// TIA Portal V16 export
// export: Created 2022-11-14T17:35:47.4589273Z, ExportSetting WithDefaults, DisplayName Totally Integrated Automation Portal, DisplayVersion V16, DisplayName TIA Portal Version Control Interface, DisplayVersion V16, DisplayName TIA Portal Openness, DisplayVersion V16, DisplayName STEP 7 Professional, DisplayVersion V16, DisplayName STEP 7 Safety, DisplayVersion V16, DisplayName WinCC Advanced, DisplayVersion V16
DATA_BLOCK "DB239_Program11"   // DB239
{ S7_Optimized_Access := 'FALSE' }
AUTHOR : Robopac
VERSION : 0.0
// stored: AutoNumber false, IsOnlyStoredInLoadMemory false, IsWriteProtectedInAS false
   VAR RETAIN
      Program11 { S7_SetPoint := 'True'} : "DatiProgramma";
   END_VAR
BEGIN
   Program11.Wrapping := TRUE;
   Program11.TopLenght := 500;
   Program11.TopRelease := 0;
   Program11.TopDown := 0;
   Program11.Top := 4;
   Program11.PressurePTime := 0;
   Program11.LifterTime := 0;
   Program11.RevOverContrast := 1;
   Program11.RopeEndCycle := 16#02;
   Program11.Spare4 := 16#01;
   Program11.RopeTime := 1500;
   Program11.RevOverClamp := 1;
   Program11.FilmForceFinalRev := 10;
   Program11.FilmPrestretchFinalRev := 100;
   Program11.ArmSpeed := 100;
   Program11.CarriageDown4Top := 500;
   Program11.TopDownTime := 1500;
   Program11.LapsUnderTop := 0;
   Program11.Spare6 := 0;
   Program11.Spare7 := 0;
   Program11.Spare8 := 0;
   Program11.Spare9 := 0;
   Program11.Spare10 := 0;
   Program11.Spare11 := 0;
   Program11.Spare12 := 0;
   Program11.Overlap0_1 := 0;
   Program11.Height1 := 130;
   Program11.Landmark1 := FALSE;
   Program11.Lifter1 := FALSE;
   Program11.SpareBit1H1 := FALSE;
   Program11.Airblower1 := TRUE;
   Program11.NextStep1 := TRUE;
   Program11.PressureP1 := TRUE;
   Program11.SpareByte2H1 := 16#00;
   Program11.Revolution1 := 1;
   Program11.RopeUnit1_1 := 16#01;
   Program11.RopeUnit1_2 := 16#01;
   Program11.FilmForce1 := 5;
   Program11.FilmPrestretch1 := 200;
   Program11.Spare3H1 := 0;
   Program11.Spare49 := 0;
   Program11.Spare50 := 0;
   Program11.Spare51 := 0;
   Program11.Spare52 := 0;
   Program11.Spare53 := 0;
   Program11.Overlap1_2 := 0;
   Program11.Height2 := 50;
   Program11.Landmark2 := FALSE;
   Program11.Lifter2 := FALSE;
   Program11.SpareBit1H2 := FALSE;
   Program11.Airblower2 := TRUE;
   Program11.NextStep2 := TRUE;
   Program11.PressureP2 := TRUE;
   Program11.SpareByte2H2 := 16#00;
   Program11.Revolution2 := 1;
   Program11.RopeUnit2_1 := 16#01;
   Program11.RopeUnit2_2 := 16#01;
   Program11.FilmForce2 := 20;
   Program11.FilmPrestretch2 := 200;
   Program11.Spare3H2 := 0;
   Program11.Spare54 := 0;
   Program11.Spare55 := 0;
   Program11.Spare56 := 0;
   Program11.Spare57 := 0;
   Program11.Spare58 := 0;
   Program11.Overlap2_3 := 100;
   Program11.Height3 := -50;
   Program11.Landmark3 := TRUE;
   Program11.Lifter3 := FALSE;
   Program11.SpareBit1H3 := FALSE;
   Program11.Airblower3 := TRUE;
   Program11.NextStep3 := TRUE;
   Program11.PressureP3 := TRUE;
   Program11.SpareByte2H3 := 16#00;
   Program11.Revolution3 := 2;
   Program11.RopeUnit3_1 := 16#01;
   Program11.RopeUnit3_2 := 16#01;
   Program11.FilmForce3 := 30;
   Program11.FilmPrestretch3 := 200;
   Program11.Spare3H3 := 0;
   Program11.Spare59 := 0;
   Program11.Spare60 := 0;
   Program11.Spare61 := 380;
   Program11.Spare62 := 2800;
   Program11.Spare63 := 0;
   Program11.Overlap3_4 := 100;
   Program11.Height4 := 100;
   Program11.Landmark4 := FALSE;
   Program11.Lifter4 := FALSE;
   Program11.SpareBit1H4 := FALSE;
   Program11.Airblower4 := TRUE;
   Program11.NextStep4 := TRUE;
   Program11.PressureP4 := TRUE;
   Program11.SpareByte2H4 := 16#00;
   Program11.Revolution4 := 3;
   Program11.RopeUnit4_1 := 16#02;
   Program11.RopeUnit4_2 := 16#02;
   Program11.FilmForce4 := 30;
   Program11.FilmPrestretch4 := 200;
   Program11.Spare3H4 := 0;
   Program11.Spare64 := 0;
   Program11.Spare65 := 0;
   Program11.Spare66 := 0;
   Program11.Spare67 := 0;
   Program11.Spare68 := 0;
   Program11.Overlap4_5 := 0;
   Program11.Height5 := 50;
   Program11.Landmark5 := FALSE;
   Program11.Lifter5 := FALSE;
   Program11.SpareBit1H5 := FALSE;
   Program11.Airblower5 := TRUE;
   Program11.NextStep5 := FALSE;
   Program11.PressureP5 := FALSE;
   Program11.SpareByte2H5 := 16#00;
   Program11.Revolution5 := 1;
   Program11.RopeUnit5_1 := 16#01;
   Program11.RopeUnit5_2 := 16#01;
   Program11.FilmForce5 := 30;
   Program11.FilmPrestretch5 := 200;
   Program11.Spare3H5 := 0;
   Program11.Spare69 := 0;
   Program11.Spare70 := 0;
   Program11.Spare71 := 0;
   Program11.Spare72 := 0;
   Program11.Spare73 := 0;
   Program11.Overlap5_6 := 100;
   Program11.Height6 := 50;
   Program11.Landmark6 := FALSE;
   Program11.Lifter6 := FALSE;
   Program11.SpareBit1H6 := FALSE;
   Program11.Airblower6 := TRUE;
   Program11.NextStep6 := FALSE;
   Program11.PressureP6 := FALSE;
   Program11.SpareByte2H6 := 16#00;
   Program11.Revolution6 := 2;
   Program11.RopeUnit6_1 := 16#02;
   Program11.RopeUnit6_2 := 16#01;
   Program11.FilmForce6 := 20;
   Program11.FilmPrestretch6 := 200;
   Program11.Spare3H6 := 0;
   Program11.Spare74 := 0;
   Program11.Spare75 := 0;
   Program11.Spare76 := 0;
   Program11.Spare77 := 0;
   Program11.Spare78 := 0;
   Program11.Overlap6_7 := 0;
   Program11.Height7 := 0;
   Program11.Landmark7 := FALSE;
   Program11.Lifter7 := FALSE;
   Program11.SpareBit1H7 := FALSE;
   Program11.Airblower7 := FALSE;
   Program11.NextStep7 := TRUE;
   Program11.PressureP7 := FALSE;
   Program11.SpareByte2H7 := 16#00;
   Program11.Revolution7 := 1;
   Program11.RopeUnit7_1 := 16#01;
   Program11.RopeUnit7_2 := 16#01;
   Program11.FilmForce7 := 0;
   Program11.FilmPrestretch7 := 100;
   Program11.Spare3H7 := 0;
   Program11.Spare79 := 0;
   Program11.Spare80 := 0;
   Program11.Spare81 := 0;
   Program11.Spare82 := 0;
   Program11.Spare83 := 0;
   Program11.Overlap7_8 := 0;
   Program11.Height8 := 0;
   Program11.Landmark8 := FALSE;
   Program11.Lifter8 := FALSE;
   Program11.SpareBit1H8 := FALSE;
   Program11.Airblower8 := FALSE;
   Program11.NextStep8 := TRUE;
   Program11.PressureP8 := FALSE;
   Program11.SpareByte2H8 := 16#00;
   Program11.Revolution8 := 1;
   Program11.RopeUnit8_1 := 16#01;
   Program11.RopeUnit8_2 := 16#01;
   Program11.FilmForce8 := 0;
   Program11.FilmPrestretch8 := 100;
   Program11.Spare3H8 := 0;
   Program11.Spare84 := 0;
   Program11.Spare85 := 0;
   Program11.Spare86 := 0;
   Program11.Spare87 := 0;
   Program11.Spare88 := 0;
   Program11.Overlap8_9 := 0;
   Program11.Height9 := 0;
   Program11.Landmark9 := FALSE;
   Program11.Lifter9 := FALSE;
   Program11.SpareBit1H9 := FALSE;
   Program11.Airblower9 := FALSE;
   Program11.NextStep9 := TRUE;
   Program11.PressureP9 := FALSE;
   Program11.SpareByte2H9 := 16#00;
   Program11.Revolution9 := 1;
   Program11.RopeUnit9_1 := 16#01;
   Program11.RopeUnit9_2 := 16#01;
   Program11.FilmForce9 := 0;
   Program11.FilmPrestretch9 := 100;
   Program11.Spare3H9 := 0;
   Program11.Spare89 := 0;
   Program11.Spare90 := 0;
   Program11.Spare91 := 0;
   Program11.Spare92 := 0;
   Program11.Spare93 := 0;
   Program11.Overlap9_10 := 0;
   Program11.Height10 := 0;
   Program11.Landmark10 := FALSE;
   Program11.Lifter10 := FALSE;
   Program11.SpareBit1H10 := FALSE;
   Program11.Airblower10 := FALSE;
   Program11.NextStep10 := FALSE;
   Program11.PressureP10 := FALSE;
   Program11.SpareByte2H10 := 16#00;
   Program11.Revolution10 := 1;
   Program11.RopeUnit10_1 := 16#01;
   Program11.RopeUnit10_2 := 16#01;
   Program11.FilmForce10 := 0;
   Program11.FilmPrestretch10 := 100;
   Program11.Spare3H10 := 0;
   Program11.Spare94 := 0;
   Program11.Spare95 := 0;
   Program11.Spare96 := 0;
   Program11.Spare97 := 0;
   Program11.Spare98 := 0;
   Program11.Overlap10_11 := 0;
   Program11.Height11 := 0;
   Program11.Landmark11 := FALSE;
   Program11.Lifter11 := FALSE;
   Program11.SpareBit1H11 := FALSE;
   Program11.Airblower11 := FALSE;
   Program11.NextStep11 := TRUE;
   Program11.PressureP11 := FALSE;
   Program11.SpareByte2H11 := 16#00;
   Program11.Revolution11 := 1;
   Program11.RopeUnit11_1 := 16#01;
   Program11.RopeUnit11_2 := 16#01;
   Program11.FilmForce11 := 0;
   Program11.FilmPrestretch11 := 100;
   Program11.Spare3H11 := 0;
   Program11.Spare99 := 0;
   Program11.Spare100 := 0;
   Program11.Spare101 := 0;
   Program11.Spare102 := 0;
   Program11.Spare103 := 0;
   Program11.Overlap11_12 := 0;
   Program11.Height12 := 0;
   Program11.Landmark12 := FALSE;
   Program11.Lifter12 := FALSE;
   Program11.SpareBit1H12 := FALSE;
   Program11.Airblower12 := FALSE;
   Program11.NextStep12 := FALSE;
   Program11.PressureP12 := FALSE;
   Program11.SpareByte2H12 := 16#00;
   Program11.Revolution12 := 1;
   Program11.RopeUnit12_1 := 16#01;
   Program11.RopeUnit12_2 := 16#01;
   Program11.FilmForce12 := 0;
   Program11.FilmPrestretch12 := 100;
   Program11.Spare3H12 := 0;
   Program11.Spare104 := 0;
   Program11.Spare105 := 0;
   Program11.Spare106 := 0;
   Program11.Spare107 := 0;
   Program11.Spare108 := 0;
END_DATA_BLOCK
